// TIA Portal V20 export
// export: Created 2025-12-01T14:57:25.5322754Z, ExportSetting None, DisplayName Totally Integrated Automation Portal, DisplayVersion V20 Update 3, DisplayName TIA Portal Openness, DisplayVersion V20 Update 3, DisplayName TIA Portal Version Control Interface, DisplayVersion V20 Update 3, DisplayName STEP 7 Professional, DisplayVersion V20 Update 3, DisplayName STEP 7 Safety, DisplayVersion V20 Update 2, DisplayName WinCC Basic/Comfort/Advanced, DisplayVersion V20 Update 3, DisplayName WinCC Professional, DisplayVersion V20 Update 3, DisplayName WinCC Unified, DisplayVersion V20 Update 3
FUNCTION_BLOCK "FB484_Interlock_IKPAL_Cajas"   // FB484, LAD
{ S7_Optimized_Access := 'FALSE' }
// stored: AutoNumber false, SetENOAutomatically false
   VAR_INPUT
      MesaCajas : UInt;
      Dir_Inicial : UInt;
      Nodo_OK : Bool;
      AvisoCajas_PRV : Bool;
   END_VAR
   VAR_OUTPUT
      EstadoIKPAL : "EstadoZona";
      PermisoCajas_PRV : Bool;
      FinCajas_PRV : Bool;
   END_VAR
   VAR
      IKPAL_PLC { S7_SetPoint := 'True'} : "Interlock_Cajas_IKPAL_PLC";
      PLC_IKPAL { S7_SetPoint := 'True'} : "Interlock_Cajas_PLC_IKPAL";
      TIM_KeepAlive { S7_SetPoint := 'True'} : TON_TIME;
      MemoKeepAlive : Bool;
   END_VAR
   VAR_TEMP
      EstadoMesaCajas : "EstadoZona";
      EstadoVIMesaCajas : "EstadosMesa";
      Guardar_AR1 : DWord;
      Guardar_AR2 : DWord;
      Interlock_Entradas : "Interlock_Cajas_IKPAL_PLC";
      Interlock_Salidas : "Interlock_Cajas_PLC_IKPAL";
      P_Entradas : Any;
      P_Salidas : Any;
      P_L_Entradas : Any;
      P_L_Salidas : Any;
      P_DI_Entradas : Any;
      P_DI_Salidas : Any;
      P_AnyTemporal : Any;
      P_Temporal : DWord;
      DBInstancia : UInt;
      LongEntradas : UInt;
      LongSalidas : UInt;
      ReturnValor : Int;
      Cero : Byte;
      FlancoKeepAlive : Bool;
   END_VAR
   VAR_TEMP   // added for the SCL form of the ladder/FBD networks
      _w1 : Bool;
      _w2 : Bool;
   END_VAR
BEGIN

REGION Network 1: INICIALIZAR
END_REGION

REGION Network 2: INICIALIZAR - Recoger las Variables de Estado de la Mesa de Preformado
   // Se recoge - Estado_CBx
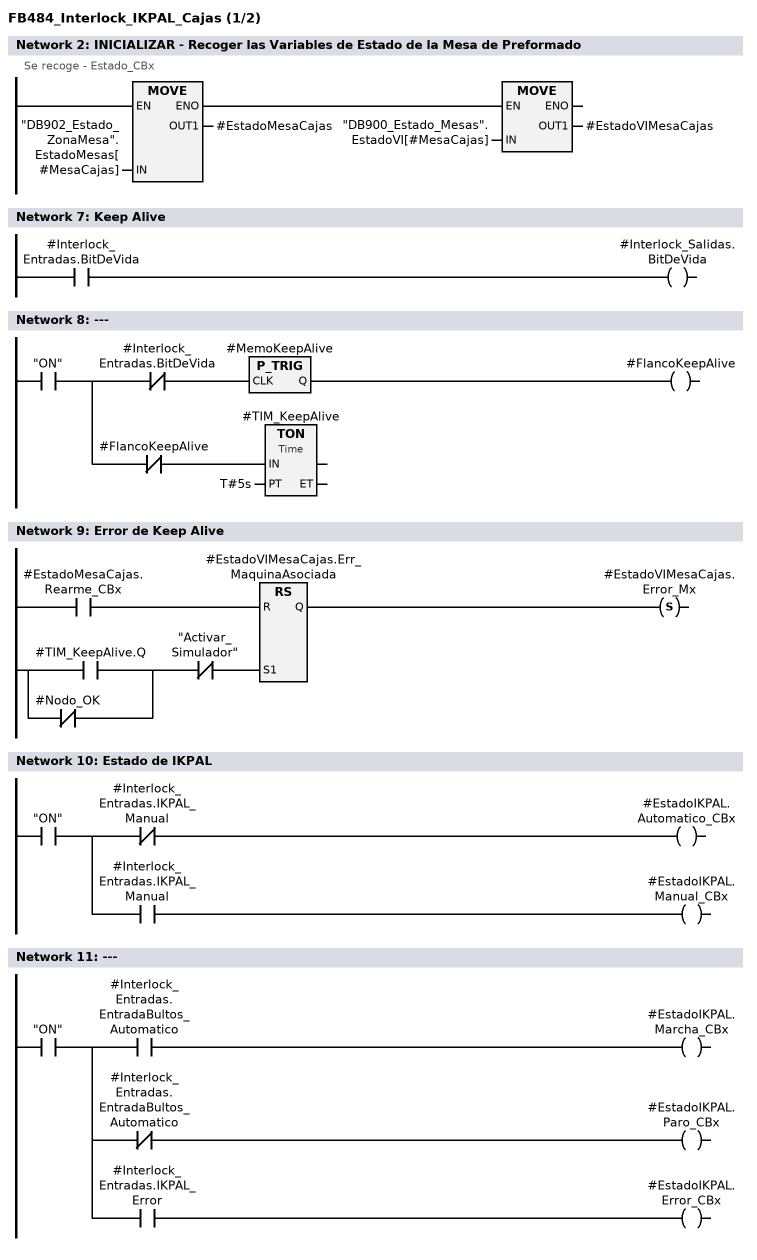
   RUNG wire#powerrail
      Move(in := "DB902_Estado_ZonaMesa".EstadoMesas[#MesaCajas], out1 => #EstadoMesaCajas)
      Move(in := "DB900_Estado_Mesas".EstadoVI[#MesaCajas], out1 => #EstadoVIMesaCajas)
   END_RUNG
   // the same network as SCL:
   #EstadoMesaCajas := "DB902_Estado_ZonaMesa".EstadoMesas[#MesaCajas];
   #EstadoVIMesaCajas := "DB900_Estado_Mesas".EstadoVI[#MesaCajas];
END_REGION

NETWORK
TITLE = Inicializar Variables Internas del Programa
//////////////////////////////////////////////////////////////////////////////
/// Inicializar las variables que necesita la FB

      L     6;  // Longitud de las Entradas
      T     #LongEntradas;
      L     6;  // Longitud de las Salidas
      T     #LongSalidas;

      L     DINO;  // Numero del DB de Instancia
      T     #DBInstancia;



NETWORK
TITLE = Preparacion de Punteros Any de las Entradas y Salidas
//////////////////////////////////////////////////////////////////////////////

      TAR1  #Guardar_AR1;  // Guardar AR1


//////////////////////////////////////////////////////////////////////////////
/// Puntero Any a las Entradas y Salidas (Temporales)

      LAR1  P##P_L_Entradas;  // - Any - Entradas del interlock
      L     B#16#10;  //   10H para S7
      T     LB [AR1, P#0.0];
      L     B#16#2;  //   Tipo de Datos (BYTE)
      T     LB [AR1, P#1.0];
      L     #LongEntradas;  //   Cantidad de datos
      T     LW [AR1, P#2.0];
      L     0;  //   Numero de DB (Temporal = 0)
      T     LW [AR1, P#4.0];
      L     P##Interlock_Entradas;  //   Direccion de Inicio
      T     LD [AR1, P#6.0];
      L     B#16#87;  //   El Area de Memoria = Temporal (Nota: No 86)
      T     LB [AR1, P#6.0];


      LAR1  P##P_L_Salidas;  // - Any - Salidas del interlock
      L     B#16#10;  //   10H para S7
      T     LB [AR1, P#0.0];
      L     B#16#2;  //   Tipo de Datos (BYTE)
      T     LB [AR1, P#1.0];
      L     #LongSalidas;  //   Cantidad de datos
      T     LW [AR1, P#2.0];
      L     0;  //   Numero de DB (Temporal = 0)
      T     LW [AR1, P#4.0];
      L     P##Interlock_Salidas;  //   Direccion de Inicio
      T     LD [AR1, P#6.0];
      L     B#16#87;  //   El Area de Memoria = Temporal (Nota: No 86)
      T     LB [AR1, P#6.0];


//////////////////////////////////////////////////////////////////////////////
/// Puntero Any a las Entradas y Salidas (DB de Instancia)

      LAR1  P##P_DI_Entradas;  // - Any - Entradas del interlock
      L     B#16#10;  //   10H para S7
      T     LB [AR1, P#0.0];
      L     B#16#2;  //   Tipo de Datos (BYTE)
      T     LB [AR1, P#1.0];
      L     #LongEntradas;  //   Cantidad de datos
      T     LW [AR1, P#2.0];
      L     #DBInstancia;  //   Numero de DB de Instancia
      T     LW [AR1, P#4.0];
      L     P##IKPAL_PLC;  //   Direccion de Inicio
      T     LD [AR1, P#6.0];
      L     B#16#84;  //   El Area de Memoria = DB Instancia
      T     LB [AR1, P#6.0];

      LAR1  P##P_DI_Salidas;  // - Any - Salidas del interlock
      L     B#16#10;  //   10H para S7
      T     LB [AR1, P#0.0];
      L     B#16#2;  //   Tipo de Datos (BYTE)
      T     LB [AR1, P#1.0];
      L     #LongSalidas;  //   Cantidad de datos
      T     LW [AR1, P#2.0];
      L     #DBInstancia;  //   Numero de DB de Instancia
      T     LW [AR1, P#4.0];
      L     P##PLC_IKPAL;  //   Direccion de Inicio
      T     LD [AR1, P#6.0];
      L     B#16#84;  //   El Area de Memoria = DB Instancia
      T     LB [AR1, P#6.0];


//////////////////////////////////////////////////////////////////////////////
/// Puntero Any - De Lectura y Escritura de QUBIQA

      LAR1  P##P_Entradas;  // - Any - Entradas del interlock
      L     B#16#10;  //   10H para S7
      T     LB [AR1, P#0.0];
      L     B#16#2;  //   Tipo de Datos (BYTE)
      T     LB [AR1, P#1.0];
      L     #LongEntradas;  //   Cantidad de datos
      T     LW [AR1, P#2.0];
      L     0;  //   Numero de DB (Temporal = 0)
      T     LW [AR1, P#4.0];
      L     #Dir_Inicial;  //   Direccion de Inicio
      SLD   3;
      T     LD [AR1, P#6.0];
      L     B#16#81;  //   El Area de Memoria = Entradas
      T     LB [AR1, P#6.0];

      LAR1  P##P_Salidas;  // - Any - Entradas del interlock
      L     B#16#10;  //   10H para S7
      T     LB [AR1, P#0.0];
      L     B#16#2;  //   Tipo de Datos (BYTE)
      T     LB [AR1, P#1.0];
      L     #LongSalidas;  //   Cantidad de datos
      T     LW [AR1, P#2.0];
      L     0;  //   Numero de DB (Temporal = 0)
      T     LW [AR1, P#4.0];
      L     #Dir_Inicial;  //   Direccion de Inicio
      SLD   3;
      T     LD [AR1, P#6.0];
      L     B#16#82;  //   El Area de Memoria = Salidas
      T     LB [AR1, P#6.0];

//////////////////////////////////////////////////////////////////////////////

      LAR1  #Guardar_AR1;  // Recuperar AR1



NETWORK
TITLE = Inicializacion de las Entradas y Salidas
//////////////////////////////////////////////////////////////////////////////
/// Inicializar el interlock (Variables Temporales)

      L     0;
      T     #Cero;

      CALL  FILL
      ( BVAL    := #Cero,
        RET_VAL := #ReturnValor,
        BLK     := #P_L_Entradas
      );  // Inicializo las Entradas

      CALL  FILL
      ( BVAL    := #Cero,
        RET_VAL := #ReturnValor,
        BLK     := #P_L_Salidas
      );  // Inicializo las Salidas



NETWORK
TITLE = Lectura de las Entradas
//////////////////////////////////////////////////////////////////////////////
/// Lectura de las Entradas

      SET;  // Comprobacion del Nodo
      AN    #Nodo_OK;
      JC    NoLeerInterlock;

      CALL  UBLKMOV
      ( SRCBLK  := #P_Entradas,
        RET_VAL := #ReturnValor,
        DSTBLK  := #P_L_Entradas
      );


//////////////////////////////////////////////////////////////////////////////
/// Final Lectura de las Entradas

NoLeerInterlock:NOP   0;

      CALL  UBLKMOV
      ( SRCBLK  := #P_L_Entradas,
        RET_VAL := #ReturnValor,
        DSTBLK  := #P_DI_Entradas
      );  // Guardar el DB de Instancia



REGION Network 7: Keep Alive
   RUNG wire#powerrail
      Contact( #Interlock_Entradas.BitDeVida )
      Coil( #Interlock_Salidas.BitDeVida )
   END_RUNG
   // the same network as SCL:
   #Interlock_Salidas.BitDeVida := #Interlock_Entradas.BitDeVida;
END_REGION

REGION Network 8: ---
   RUNG wire#powerrail
      Contact( "ON" )
      wire#w1
      I_Contact( #Interlock_Entradas.BitDeVida )
      P_Trig( #MemoKeepAlive )
      Coil( #FlancoKeepAlive )
   END_RUNG
   RUNG wire#w1
      I_Contact( #FlancoKeepAlive )
      { S7_Templates := "time_type := Time" } #TIM_KeepAlive.TON(pt := T#5s, et =>)
   END_RUNG
   // the same network as SCL:
   #_w1 := "ON" AND NOT #Interlock_Entradas.BitDeVida;
   #_w2 := #_w1 AND NOT #MemoKeepAlive;   // rising edge
   #MemoKeepAlive := #_w1;
   #FlancoKeepAlive := #_w2;
   #TIM_KeepAlive(IN := "ON" AND NOT #FlancoKeepAlive, PT := T#5s);   // TON
END_REGION

REGION Network 9: Error de Keep Alive
   RUNG wire#powerrail
      Contact( #EstadoMesaCajas.Rearme_CBx )
      S_RS(operand := #EstadoVIMesaCajas.Err_MaquinaAsociada, s1 := wire#w2)
      S_Coil( #EstadoVIMesaCajas.Error_Mx )
   END_RUNG
   RUNG wire#powerrail
      Contact( #TIM_KeepAlive.Q )
      wire#w1
      I_Contact( "Activar_Simulador" )
   END_RUNG wire#w2
   RUNG wire#powerrail
      I_Contact( #Nodo_OK )
   END_RUNG wire#w1
   // the same network as SCL:
   IF #EstadoMesaCajas.Rearme_CBx THEN
       #EstadoVIMesaCajas.Err_MaquinaAsociada := FALSE;   // RS flip-flop
   END_IF;
   IF (#TIM_KeepAlive.Q OR NOT #Nodo_OK) AND NOT "Activar_Simulador" THEN
       #EstadoVIMesaCajas.Err_MaquinaAsociada := TRUE;
   END_IF;
   IF #EstadoVIMesaCajas.Err_MaquinaAsociada THEN #EstadoVIMesaCajas.Error_Mx := TRUE; END_IF;
END_REGION

REGION Network 10: Estado de IKPAL
   RUNG wire#powerrail
      Contact( "ON" )
      wire#w1
      I_Contact( #Interlock_Entradas.IKPAL_Manual )
      Coil( #EstadoIKPAL.Automatico_CBx )
   END_RUNG
   RUNG wire#w1
      Contact( #Interlock_Entradas.IKPAL_Manual )
      Coil( #EstadoIKPAL.Manual_CBx )
   END_RUNG
   // the same network as SCL:
   #EstadoIKPAL.Automatico_CBx := "ON" AND NOT #Interlock_Entradas.IKPAL_Manual;
   #EstadoIKPAL.Manual_CBx := "ON" AND #Interlock_Entradas.IKPAL_Manual;
END_REGION

REGION Network 11: ---
   RUNG wire#powerrail
      Contact( "ON" )
      wire#w1
      Contact( #Interlock_Entradas.EntradaBultos_Automatico )
      Coil( #EstadoIKPAL.Marcha_CBx )
   END_RUNG
   RUNG wire#w1
      I_Contact( #Interlock_Entradas.EntradaBultos_Automatico )
      Coil( #EstadoIKPAL.Paro_CBx )
   END_RUNG
   RUNG wire#w1
      Contact( #Interlock_Entradas.IKPAL_Error )
      Coil( #EstadoIKPAL.Error_CBx )
   END_RUNG
   // the same network as SCL:
   #EstadoIKPAL.Marcha_CBx := "ON" AND #Interlock_Entradas.EntradaBultos_Automatico;
   #EstadoIKPAL.Paro_CBx := "ON" AND NOT #Interlock_Entradas.EntradaBultos_Automatico;
   #EstadoIKPAL.Error_CBx := "ON" AND #Interlock_Entradas.IKPAL_Error;
END_REGION

REGION Network 12: Estado de la Mesa de Cajas
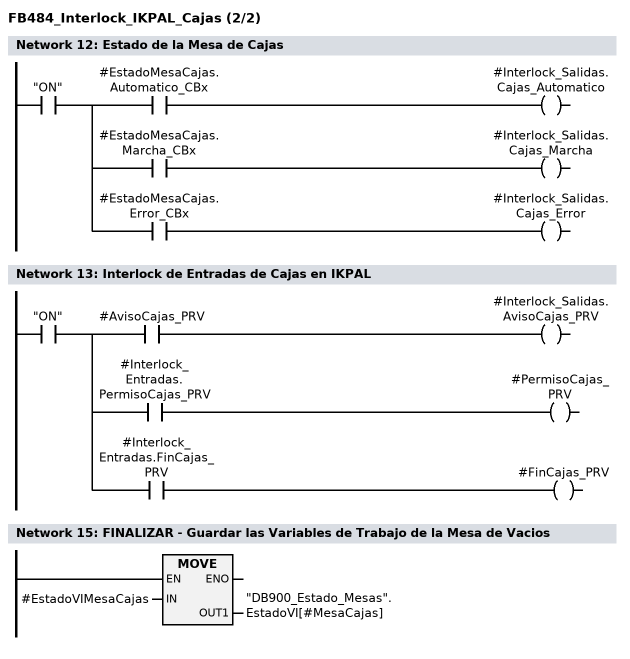
   RUNG wire#powerrail
      Contact( "ON" )
      wire#w1
      Contact( #EstadoMesaCajas.Automatico_CBx )
      Coil( #Interlock_Salidas.Cajas_Automatico )
   END_RUNG
   RUNG wire#w1
      Contact( #EstadoMesaCajas.Marcha_CBx )
      Coil( #Interlock_Salidas.Cajas_Marcha )
   END_RUNG
   RUNG wire#w1
      Contact( #EstadoMesaCajas.Error_CBx )
      Coil( #Interlock_Salidas.Cajas_Error )
   END_RUNG
   // the same network as SCL:
   #Interlock_Salidas.Cajas_Automatico := "ON" AND #EstadoMesaCajas.Automatico_CBx;
   #Interlock_Salidas.Cajas_Marcha := "ON" AND #EstadoMesaCajas.Marcha_CBx;
   #Interlock_Salidas.Cajas_Error := "ON" AND #EstadoMesaCajas.Error_CBx;
END_REGION

REGION Network 13: Interlock de Entradas de Cajas en IKPAL
   RUNG wire#powerrail
      Contact( "ON" )
      wire#w1
      Contact( #AvisoCajas_PRV )
      Coil( #Interlock_Salidas.AvisoCajas_PRV )
   END_RUNG
   RUNG wire#w1
      Contact( #Interlock_Entradas.PermisoCajas_PRV )
      Coil( #PermisoCajas_PRV )
   END_RUNG
   RUNG wire#w1
      Contact( #Interlock_Entradas.FinCajas_PRV )
      Coil( #FinCajas_PRV )
   END_RUNG
   // the same network as SCL:
   #Interlock_Salidas.AvisoCajas_PRV := "ON" AND #AvisoCajas_PRV;
   #PermisoCajas_PRV := "ON" AND #Interlock_Entradas.PermisoCajas_PRV;
   #FinCajas_PRV := "ON" AND #Interlock_Entradas.FinCajas_PRV;
END_REGION

NETWORK
TITLE = Escritura de las Salidas
//////////////////////////////////////////////////////////////////////////////
/// Escritura de las Salidas

      SET;  // Comprobacion del Nodo
      AN    #Nodo_OK;
      JC    NoEscribirInterlock;

      CALL  UBLKMOV
      ( SRCBLK  := #P_L_Salidas,
        RET_VAL := #ReturnValor,
        DSTBLK  := #P_Salidas
      );


//////////////////////////////////////////////////////////////////////////////
/// Final Esctitura de las Salidas

NoEscribirInterlock:NOP   0;

      CALL  UBLKMOV
      ( SRCBLK  := #P_L_Salidas,
        RET_VAL := #ReturnValor,
        DSTBLK  := #P_DI_Salidas
      );  // Guardar el DB de Instancia




REGION Network 15: FINALIZAR - Guardar las Variables de Trabajo de la Mesa de Vacios
   RUNG wire#powerrail
      Move(in := #EstadoVIMesaCajas, out1 => "DB900_Estado_Mesas".EstadoVI[#MesaCajas])
   END_RUNG
   // the same network as SCL:
   "DB900_Estado_Mesas".EstadoVI[#MesaCajas] := #EstadoVIMesaCajas;
END_REGION
END_FUNCTION_BLOCK
